FUNCTION RESET_ZONA_INPUT : ZONA_INPUT

VAR_INPUT
	INPUT : ZONA_INPUT;
END_VAR

VAR_OUTPUT
	OUTPUT : ZONA_INPUT;
END_VAR

INPUT.ENABLE := FALSE;
INPUT.RIPRISTINO := FALSE;
INPUT.LIBERO := FALSE;
INPUT.TRIGGER := FALSE;
OUTPUT := INPUT;

END_FUNCTION

(* stored: Version 1.1.0.1, ProductVersion 3.1.4024.12
   POU RESET_ZONA_INPUT: Id {3fdce18d-55df-45a4-8cca-3f2af29fe009}, SpecialFunc None *)
